PROGRAM MAIN
VAR
	sIpAddr : STRING[15] := '192.168.001.252';
	nport : UINT := 502;
	nUnitID : BYTE := 1;
	tTimeOut : TIME := T#1S;
	nOfReg : UINT := 10;
	nAddr :WORD := 0;
	
	fb_MBReadRegister: FB_MBReadRegs;
	bReadEnable: BOOL;
	bReadBusyFlag: BOOL;
	bReadErrorFlag: BOOL;
	nReadErrorID: UDINT;
	ireadReg : ARRAY[1..10] OF WORD;
	
	n :INT := 0;
	
	bWriteBusyFlag: BOOL;
	bWriteEnable: BOOL;
	fb_MBWriteRegister: FB_MBWriteRegs;
	bWriteErrorFlag: BOOL;
	nWriteErrorID: UDINT;
	iWriteReg : ARRAY[1..10] OF WORD;

END_VAR

(* Version history: 
Date          | Version    | created under        | Author          | Remark 
---------------------------------------------------------------------------------------- 
20/06/2022    | 1.0.0      | V3.1 (Build 4024.29) | Gokul G         | first release 
	* Basic Modbus TCP/IP Register Read/Write 
	
*) 
(* Modbus TCP/IP Communication  
1.First Install TF6250 Software in both Target & Enginnering PC Add Tc2_ModbusSrv Library 
2.In Main Program
	Variable 
	sIpAddr : STRING[15] := '192.168.001.252';
	nport : UINT := 502;
	nUnitID : BYTE := 1;
	tTimeOut : TIME := T#1S;
	nOfReg : UINT := 10;
	nAddr :WORD := 0;
	
	fb_MBReadRegister: FB_MBReadRegs;
	bReadEnable: BOOL;
	bReadBusyFlag: BOOL;
	bReadErrorFlag: BOOL;
	nReadErrorID: UDINT;
	ireadReg : ARRAY[1..10] OF WORD;
	
	n :INT := 0;
	
	bWriteBusyFlag: BOOL;
	bWriteEnable: BOOL;
	fb_MBWriteRegister: FB_MBWriteRegs;
	bWriteErrorFlag: BOOL;
	nWriteErrorID: UDINT;
	iWriteReg : ARRAY[1..10] OF WORD;
	
	Program 
	(* For Alternate Read & Write of Register *)
	IF n >= 100 AND NOT bReadBusyFlag THEN
		bReadEnable := TRUE;
	ELSIF n >= 200 AND NOT bWriteBusyFlag THEN
		bWriteEnable := TRUE;
		n := 0;
	END_IF
	n := n+1;

	(* Read Register *)
	fb_MBReadRegister(
		sIPAddr:= sIpAddr, 
		nTCPPort:= nport,
		nUnitID:= nUnitID, 
		nQuantity:= nOfReg , 
		nMBAddr:= nAddr , 
		cbLength:= SIZEOF(ireadReg), 
		pDestAddr:=ADR(ireadReg) , 
		bExecute:=bReadEnable , 
		tTimeout:= tTimeOut , 
		bBusy=> bReadBusyFlag, 
		bError=> bReadErrorFlag , 
		nErrId=> nReadErrorID , 
		cbRead=> );
	bReadEnable := FALSE;
	
	(* Write Register *)
	fb_MBWriteRegister(
		sIPAddr:= sIpAddr, 
		nTCPPort:= nport , 
		nUnitID:= nUnitID , 
		nQuantity:= nOfReg, 
		nMBAddr:= nAddr + 10 , 
		cbLength:= SIZEOF(iWriteReg), 
		pSrcAddr:= ADR(iWriteReg), 
		bExecute:= bWriteEnable, 
		tTimeout:= tTimeOut, 
		bBusy=> bWriteBusyFlag, 
		bError=> bWriteErrorFlag, 
		nErrId=> nWriteErrorID );	
	bWriteEnable := FALSE;
3.Set IP Adress of Servers as per requirement & port should be specified (Usally 502 but it can be changed if multiple modbus servers are there in same IP)
4.Program will alternately read & write register every 1 secs

Note :
	If Address in Modscan is 1 then in MBAddress it should be 0 (-1)
	
*)

(* For Alternate Read & Write of Register *)
IF n >= 100 AND NOT bReadBusyFlag THEN
	bReadEnable := TRUE;
ELSIF n >= 200 AND NOT bWriteBusyFlag THEN
	bWriteEnable := TRUE;
	n := 0;
END_IF
n := n+1;

(* Read Register *)
fb_MBReadRegister(
	sIPAddr:= sIpAddr, 
	nTCPPort:= nport,
	nUnitID:= nUnitID, 
	nQuantity:= nOfReg , 
	nMBAddr:= nAddr , 
	cbLength:= SIZEOF(ireadReg), 
	pDestAddr:=ADR(ireadReg) , 
	bExecute:=bReadEnable , 
	tTimeout:= tTimeOut , 
	bBusy=> bReadBusyFlag, 
	bError=> bReadErrorFlag , 
	nErrId=> nReadErrorID , 
	cbRead=> );
bReadEnable := FALSE;

(* Write Register *)
fb_MBWriteRegister(
	sIPAddr:= sIpAddr, 
	nTCPPort:= nport , 
	nUnitID:= nUnitID , 
	nQuantity:= nOfReg, 
	nMBAddr:= nAddr + 10 , 
	cbLength:= SIZEOF(iWriteReg), 
	pSrcAddr:= ADR(iWriteReg), 
	bExecute:= bWriteEnable, 
	tTimeout:= tTimeOut, 
	bBusy=> bWriteBusyFlag, 
	bError=> bWriteErrorFlag, 
	nErrId=> nWriteErrorID );	
bWriteEnable := FALSE;

END_PROGRAM

(* stored: Version 1.1.0.1, ProductVersion 3.1.4024.11
   POU MAIN: Id {9ea0e380-1a7b-4bd1-a863-dcc7ae2702da}, SpecialFunc None *)
